FUNCTION_BLOCK FB_ModbusSlave IMPLEMENTS I_ModbusSlave
VAR
	iUnitID			: 		BYTE;
	arrAddress		:		ARRAY [0..50] OF ARRAY [0..1] OF WORD;
	iNumAddRegion	:		UINT;
	bSwap			:		BOOL;
	
	sName			:		STRING;

END_VAR

PROPERTY Address : POINTER TO WORD
GET
Address := ADR(arrAddress);
END_GET
END_PROPERTY

METHOD Convert : BOOL
VAR_INPUT
	iRegionNo	:	INT;
	pReadData	:	POINTER TO BYTE;
END_VAR
END_METHOD

METHOD FirstCycle : BOOL
VAR_INPUT
END_VAR
END_METHOD

PROPERTY Name : STRING
GET
Name := sName;
END_GET
SET
sName := Name;
END_SET
END_PROPERTY

PROPERTY NumAddRegion : UINT
GET
NumAddRegion := iNumAddRegion;
END_GET
END_PROPERTY

PROPERTY UnitID : BYTE
GET
UnitID := iUnitID;
END_GET
SET
iUnitID := UnitID;
END_SET
END_PROPERTY

END_FUNCTION_BLOCK

(* stored: Version 1.1.0.1, ProductVersion 3.1.4024.12
   POU FB_ModbusSlave: Id {8e91e30b-c030-4324-9a58-08958f9a6361}, SpecialFunc None
   Property Address: Id {6673aa7a-a0df-48bb-86cd-95e052a71ce1}
   Get Get: Id {7029230a-5cfd-4f5f-a728-bb0ce320e832}
   Method Convert: Id {e961461b-a0b2-472d-bf52-574004f124cf}
   Method FirstCycle: Id {841c47f5-ed41-4f9d-b6e9-9d57d2118f5d}
   Property Name: Id {80691629-a680-4048-94be-bd030236c721}
   Get Get: Id {8a564c6a-458f-4500-ab50-793267d106f9}
   Set Set: Id {4e06a7ff-6002-43a5-81a3-3a4646ea8f0b}
   Property NumAddRegion: Id {6f082c03-284b-4503-a54e-c54009e2d9b4}
   Get Get: Id {d0415010-03aa-46af-bfd3-d1307c65e11d}
   Property UnitID: Id {09b40999-a093-4b5e-a633-0dac9ebd5691}
   Get Get: Id {25467e3f-4d89-4043-b689-ef798c7d8419}
   Set Set: Id {2df837ea-aa39-4110-b397-a4f53cdd7a6d} *)
